// TIA Portal V18 export
// export: Created 2025-12-01T12:38:39.8541137Z, ExportSetting None, DisplayName Totally Integrated Automation Portal, DisplayVersion V18 Update 5, DisplayName TIA Portal Openness, DisplayVersion V18 Update 5, DisplayName TIA Portal Teamcenter Gateway, DisplayVersion V18, DisplayName TIA Portal Version Control Interface, DisplayVersion V18, DisplayName STEP 7 Professional, DisplayVersion V18 Update 5, DisplayName STEP 7 Safety, DisplayVersion V18, DisplayName WinCC Professional, DisplayVersion V18 Update 5
FUNCTION_BLOCK "SevroStart&PosCheck_IAI"   // FB2209, LAD
{ S7_Optimized_Access := 'TRUE' }
// stored: AutoNumber false, MemoryReserve 100, SetENOAutomatically false
   VAR_INPUT
      iRef_Homed { ExternalAccessible := 'False'; ExternalVisible := 'False'; ExternalWritable := 'False'} : Bool;
      iStandstill { ExternalAccessible := 'False'; ExternalVisible := 'False'; ExternalWritable := 'False'} : Bool;
      iReset : Bool;
      interlcok : Bool;   // 启动互锁
      "iActual Posi" { ExternalAccessible := 'False'; ExternalVisible := 'False'; ExternalWritable := 'False'} : Real;
      "iTol+" { ExternalAccessible := 'False'; ExternalVisible := 'False'; ExternalWritable := 'False'} : Real;
      "iTol-" { ExternalAccessible := 'False'; ExternalVisible := 'False'; ExternalWritable := 'False'} : Real;
      iStartTon : Time := T#200ms;   // 启动延迟
   END_VAR
   VAR_OUTPUT
      oStartPos : Bool;   // 启动
      DoublePosError : Bool;   // 多位置触发
   END_VAR
   VAR_IN_OUT
      ioPoint : Array[0..39] of Struct
         Start : Bool;
         Achieve : Bool;
      END_STRUCT;
      ioList : "PosList_IAI";
      ioPosNumberSelect : Int;   // 位置启动
   END_VAR
   VAR
      TON : Array[0..1] of TON_TIME;
      StartCount { S7_SetPoint := 'True'} : Int;   // 启动计数
   END_VAR
   VAR_TEMP
      "Actual Posi+Tol" : Real;
      "Actual Posi-Tol" : Real;
      Index : Array[0..7] of Int;   // 位置启动
      PosStart : Bool;
   END_VAR
   VAR_TEMP   // added for the SCL form of the ladder/FBD networks
      _w1 : Bool;
   END_VAR
BEGIN

REGION Network 1 (SCL): 检查当前启动位置号
   #Index[1] := 0;
   #PosStart := false;
   FOR #Index[1] := 0 TO 39 DO
       IF #ioPoint[#Index[1]].Start THEN

           #ioPosNumberSelect := #Index[1];//当前启动位置号
           #PosStart := TRUE;
           EXIT;
       END_IF;
   END_FOR;
   #Index[2] := 0;
   #StartCount := 0;
   FOR #Index[2] := 0 TO 39 DO
       IF #ioPoint[#Index[2]].Start THEN

           #StartCount := #StartCount+1;//当前启动位置号


       END_IF;
       IF #Index[2] = 39 THEN

           EXIT;
       END_IF;

   END_FOR;
END_REGION

REGION Network 2: 位置给定
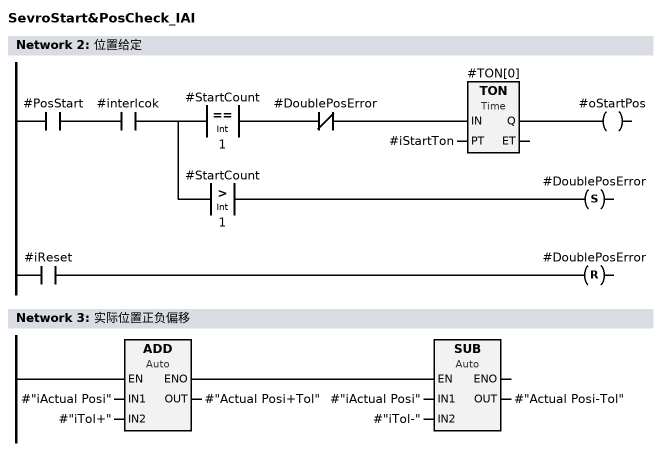
   RUNG wire#powerrail
      Contact( #PosStart )
      Contact( #interlcok )
      wire#w1
      { S7_Templates := "SrcType := Int" } EQ_Contact(in1 := #StartCount, in2 := 1)
      I_Contact( #DoublePosError )
      { S7_Templates := "time_type := Time" } #TON[0].TON(pt := #iStartTon, et =>)
      Coil( #oStartPos )
   END_RUNG
   RUNG wire#w1
      { S7_Templates := "SrcType := Int" } GT_Contact(in1 := #StartCount, in2 := 1)
      S_Coil( #DoublePosError )
   END_RUNG
   RUNG wire#powerrail
      Contact( #iReset )
      R_Coil( #DoublePosError )
   END_RUNG
   // the same network as SCL:
   #_w1 := #PosStart AND #interlcok;
   #TON[0].TON(IN := #_w1 AND (#StartCount = 1) AND NOT #DoublePosError, PT := #iStartTon);
   #oStartPos := #TON[0].Q;
   IF #_w1 AND (#StartCount > 1) THEN #DoublePosError := TRUE; END_IF;
   IF #iReset THEN #DoublePosError := FALSE; END_IF;
END_REGION

REGION Network 3: 实际位置正负偏移
   RUNG wire#powerrail
      Add(in1 := #"iActual Posi", in2 := #"iTol+", out => #"Actual Posi+Tol")
      Sub(in1 := #"iActual Posi", in2 := #"iTol-", out => #"Actual Posi-Tol")
   END_RUNG
   // the same network as SCL:
   #"Actual Posi+Tol" := #"iActual Posi" + #"iTol+";
   #"Actual Posi-Tol" := #"iActual Posi" - #"iTol-";
END_REGION

REGION Network 4 (SCL): 位置检查


   #Index[3] := 0;
   FOR #Index[3] := 0 TO 39 DO
       IF #ioList.List[ #Index[3]].Pos>= #"Actual Posi-Tol"
           AND #ioList.List[ #Index[3]].Pos<= #"Actual Posi+Tol"
       THEN
         #ioPoint[#Index[3]].Achieve := TRUE;
       ELSE
           #ioPoint[#Index[3]].Achieve := FALSE;
       END_IF;
   END_FOR;
END_REGION
END_FUNCTION_BLOCK
